// TwinCAT 3 PLC project Cappuccino_machine
// ProgramVersion: 3.1.4024.0
// libraries:
//   Tc2_Standard, * (Beckhoff Automation GmbH)
//   Tc2_System, * (Beckhoff Automation GmbH)
//   Tc3_Module, * (Beckhoff Automation GmbH)
//   VisuSymbols,3.5.10.0,System
// project tree:
//   / GlobalTextList.TcGTLO, PlcTask.TcTTO (not stored), Visualization Manager.TcVMO (not stored)
//   GVLs/ GVL.TcGVL
//   POUs/ functie.TcPOU (not stored), Proces_1.TcPOU, Proces_2.TcPOU
//   VISUs/ Visualization.TcVIS
// real-time tasks:
//   TASK PlcTask: cycle T#10ms, priority 20, ADS port 350

// ---- GVLs/GVL.TcGVL
{attribute 'qualified_only'}
VAR_GLOBAL
// Inputs			
Power_ON		: BOOL;
Water_opgewarmt	: BOOL;


// Outputs
Spoelen_machine 	: BOOL;
Water_verwarmen		: BOOL;


END_VAR

// ---- POUs/Proces_1.TcPOU
PROGRAM Proces_1
VAR
// INputs
Start			: BOOL;
Beker_aanwezig	: BOOL;
Bonen_aanwezig	: BOOL;
Melk_aanwezig	: BOOL;
Voldoende_water	: BOOL;



// Outputs
Led_ready_start		: BOOL;
Melk_verwarming		: BOOL;
Melk_pomp			: BOOL;
Bonen_malen			: BOOL;
Water_pomp			: BOOL;




Step		: UINT;	
Spoelen		: BOOL; 
Start_Spoelen :BOOL;	




// Timers
Timer 		: TON;
Timer2 		: TON;
Timer3 		: TON;
Timer4 		: TON;
END_VAR



// Statemachine
CASE Step OF
	0: //Init stap 0
		IF GVL.Power_ON = TRUE THEN
			Step				:=10;
		END_IF
	

	10: // Spoelen machine 
	Timer(IN:=TRUE, PT:=T#5S);
	Start_Spoelen := TRUE;
	Spoelen := functie(Spoelen_start := Start_Spoelen, Timer);	

	
	IF Spoelen = TRUE THEN
		Step		:=20;
	END_IF

	20: // klaar om te starten
	Timer(IN:=FALSE, PT:=T#5S);
	//spoelen := FALSE;
	IF Bonen_aanwezig = TRUE  AND Melk_aanwezig = TRUE AND Voldoende_water THEN
		Led_ready_start := TRUE;
		Step 	:= 30;
	END_IF
	
	
	30: // Wanneer beker aanwezig is en op strat word geklikt. Melk word verwarmt en bonen worden gemalen.
	IF Start = TRUE AND Beker_aanwezig = TRUE THEN
		Led_ready_start := FALSE;
		Melk_verwarming	:= TRUE;
		Bonen_malen		:= TRUE;
		Timer2(IN:=TRUE, PT:=T#5S);	
	END_IF
	
	
	IF Timer2.Q = TRUE THEN
		Timer2(IN:=FALSE);
		Start := FALSE;
		Step	:= 40;
	END_IF
	

	40: // na 5 sec gaat bonen malen uit en de melk pomp aan voor toevoegen melk.
	Bonen_malen		:= FALSE;
	Melk_pomp		:= TRUE;
	
	Timer3(IN:=TRUE, PT:=T#5S);
	
	IF Timer3.Q = TRUE THEN
		Timer3(IN:=FALSE);
		Step	:= 50;
	END_IF	
	
	50: // na 5 sec melk verwarming en pomp gaan uit. water word door de bonen gepompt.
	Melk_verwarming	:= FALSE;
	Melk_pomp		:= FALSE;
	Water_pomp		:= TRUE;
	
	Timer4(IN:=TRUE, PT:=T#5S);
	
	IF Timer4.Q = TRUE THEN
		Timer4(IN:=FALSE);
		Step	:= 60;
	END_IF

	60: 
	Water_pomp		:= FALSE;
	
	IF Beker_aanwezig = FALSE THEN
		Step	:= 10;
	END_IF
END_CASE

END_PROGRAM

// ---- POUs/Proces_2.TcPOU
PROGRAM Proces_2
VAR
	
	Step: INT;
END_VAR

CASE Step OF

0: // wachten op machine aan
IF GVL.Power_ON THEN 
	Step			:=10;
END_IF	


10: // water kan verwarmt worden
GVL.Water_verwarmen := TRUE;

IF GVL.Water_opgewarmt THEN
	Step			:=20;
END_IF

20: // water is opgewarmt. Waneer water niet meer op temperatuur is terug naar step 10
GVL.Water_verwarmen := FALSE;

IF GVL.Water_opgewarmt = FALSE THEN
	Step			:=10;
END_IF
END_CASE

END_PROGRAM

// ---- GlobalTextList.TcGTLO
TEXTLIST GlobalTextList
  78 = 'Beker aanwezig'
  494 = 'Bonen aanwezig'
  286 = 'Bonen malen'
  913 = 'Melk aanwezig'
  830 = 'Melk Pomp'
  26 = 'Melk verwarmen'
  398 = 'Power ON'
  827 = 'Ready to start'
  493 = 'Spoelen machine'
  763 = 'Start'
  86 = 'Voldoende water'
  215 = 'Water opgewarmt'
  974 = 'Water opwarmen'
  43 = 'Water Pomp'
END_TEXTLIST

// ---- VISUs/Visualization.TcVIS
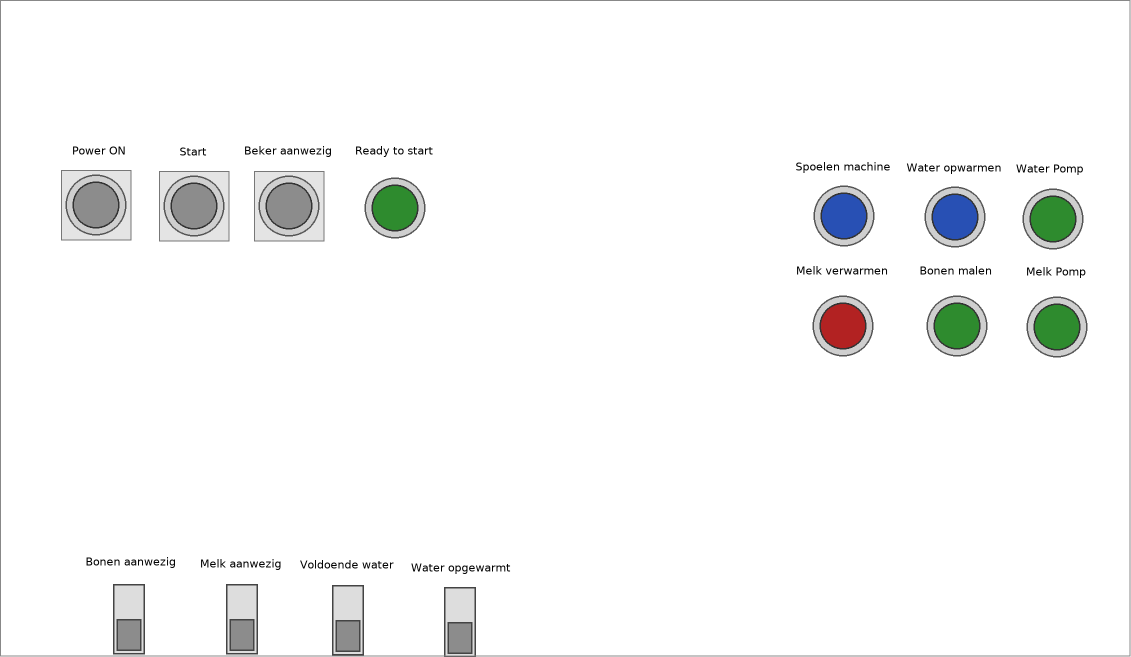
VISUALIZATION Visualization  // 1131x657
    Lamp1 (809,181 70x70), tooltip "Spoelen machine", variable: GVL.Spoelen_machine, style: Lamp-Lamp1-Blue
    PushSwitch (61,170 70x70), variable: GVL.Power_ON, behaviour: TOGGLE, style: Switch-PushSwitch-Gray
    Label (768,152 150x30), "Spoelen machine"
    Lamp1 (360,173 70x70), variable: Proces_1.Led_ready_start, style: Lamp-Lamp1-Green
    Label (319,136 150x30), "Ready to start"
    DipSwitch (94,584 70x70), variable: Proces_1.Bonen_aanwezig, behaviour: TOGGLE, style: Switch-DipSwitch-Gray
    Label (56,547 150x30), "Bonen aanwezig"
    Label (166,549 150x30), "Melk aanwezig"
    DipSwitch (207,584 70x70), variable: Proces_1.Melk_aanwezig, behaviour: TOGGLE, style: Switch-DipSwitch-Gray
    Label (272,550 150x30), "Voldoende water"
    DipSwitch (313,585 70x70), variable: Proces_1.Voldoende_water, behaviour: TOGGLE, style: Switch-DipSwitch-Gray
    Lamp1 (920,182 70x70), variable: GVL.Water_verwarmen, style: Lamp-Lamp1-Blue
    Label (879,153 150x30), "Water opwarmen"
    DipSwitch (425,587 70x70), variable: GVL.Water_opgewarmt, behaviour: TOGGLE, style: Switch-DipSwitch-Gray
    Label (386,553 150x30), "Water opgewarmt"
    Label (24,136 150x30), "Power ON"
    PushSwitch (159,171 70x70), variable: Proces_1.Start, behaviour: TOGGLE, style: Switch-PushSwitch-Gray
    Label (118,137 150x30), "Start"
    PushSwitch (254,171 70x70), variable: Proces_1.Beker_aanwezig, behaviour: TOGGLE, style: Switch-PushSwitch-Gray
    Label (213,136 150x30), "Beker aanwezig"
    Lamp1 (808,291 70x70), variable: Proces_1.Melk_verwarming, style: Lamp-Lamp1-Red
    Label (767,256 150x30), "Melk verwarmen"
    Label (981,257 150x30), "Melk Pomp"
    Lamp1 (1022,292 70x70), variable: Proces_1.Melk_pomp, style: Lamp-Lamp1-Green
    Label (881,256 150x30), "Bonen malen"
    Lamp1 (922,291 70x70), variable: Proces_1.Bonen_malen, style: Lamp-Lamp1-Green
    Lamp1 (1018,184 70x70), variable: Proces_1.Water_pomp, style: Lamp-Lamp1-Green
    Label (975,154 150x30), "Water Pomp"
END_VISUALIZATION
